// TIA Portal project "elektro_boiler" (V16)

(* hardware
DEVICE "S7-1200 station_1"  S7-1200 Station
   slot 0: "Rack_0"  S7-1200 Rack  Rack  V1.0
   slot 1: "PLC_1"  CPU 1215C DC/DC/Rly  6ES7 215-1HG40-0XB0  V4.4
   slot 2: "AI 8x13BIT_1"  6ES7 231-4HF32-0XB0  V2.1
*)

// ===== PLC "PLC_1"  CPU 1215C DC/DC/Rly =====

VAR_GLOBAL   // PLC tag table "Default tag table"
   "Clock_Byte" AT %MB0 : Byte;
   "Clock_10Hz" AT %M0.0 : Bool;
   "Clock_5Hz" AT %M0.1 : Bool;
   "Clock_2.5Hz" AT %M0.2 : Bool;
   "Clock_2Hz" AT %M0.3 : Bool;
   "Clock_1.25Hz" AT %M0.4 : Bool;
   "Clock_1Hz" AT %M0.5 : Bool;
   "Clock_0.625Hz" AT %M0.6 : Bool;
   "Clock_0.5Hz" AT %M0.7 : Bool;
   "TRUE" AT %M5.1 : Bool;
   "FALSE" AT %M5.0 : Bool;
   "puls_1_sec_t" AT %M4.0 : Bool;
   "puls_1_sec" AT %M4.1 : Bool;
   "EVEN" AT %M4.2 : Bool;
   "ODD" AT %M4.3 : Bool;
   "System_Byte" AT %MB1 : Byte;
   "FirstScan" AT %M1.0 : Bool;
   "DiagStatusUpdate" AT %M1.1 : Bool;
   "AlwaysTRUE" AT %M1.2 : Bool;
   "AlwaysFALSE" AT %M1.3 : Bool;
   "System_Byte(1)" AT %MB1 : Byte;
   "PUMP" AT %I0.0 : Bool;
   "AUTO_MAN" AT %I0.1 : Bool;
   "ELECTODE_DI1" AT %I0.2 : Bool;
   "ELECTODE_DI2" AT %I0.3 : Bool;
   "ELECTODE_DI3" AT %I0.4 : Bool;
   "ELECTODE_DI4" AT %I0.5 : Bool;
   "ELECTODE_DI5" AT %I0.6 : Bool;
   "ELECTODE_DI6" AT %I0.7 : Bool;
   "ELECTODE_DI7" AT %I1.0 : Bool;
   "ELECTODE_DI8" AT %I1.1 : Bool;
   "Tag_1" AT %Q1.1 : Bool;
   "Tag_2" AT %M6.0 : Bool;
END_VAR

VAR_GLOBAL   // PLC tag table "DO"
   "ELECTR_DO_1" AT %Q0.0 : Bool;
   "ELECTR_DO_2" AT %Q0.1 : Bool;
   "ELECTR_DO_3" AT %Q0.2 : Bool;
   "ELECTR_DO_4" AT %Q0.3 : Bool;
   "ELECTR_DO_5" AT %Q0.4 : Bool;
   "ELECTR_DO_6" AT %Q0.5 : Bool;
   "ELECTR_DO_7" AT %Q0.6 : Bool;
   "ELECTR_DO_8" AT %Q0.7 : Bool;
   "ZUMMER" AT %Q1.0 : Bool;
END_VAR

VAR_GLOBAL   // PLC tag table "AI"
   "PRESSURE" AT %IW112 : Int;
   "TEMP_IN" AT %IW114 : Int;
   "res1" AT %IW116 : Int;
   "CURRENT_A" AT %IW118 : Int;
   "CURRENT_B" AT %IW120 : Int;
   "CURRENT_C" AT %IW122 : Int;
END_VAR

TYPE "AIN"
   STRUCT
      data_raw : Int;   // Сырое значение
      signal : Real;   // Значение сигнала в электрических единицах (мА, В и т.д.)
      eng : Real;   // Масштабированное значение аналогового сигнала
      status_0 : Bool;   // Неисправность канала
      status_1 : Bool;   // Ошибка калибровки (CalFault)
      status_2 : Bool;   // Выше HH
      status_3 : Bool;   // Выше H
      status_4 : Bool;   // Ниже L
      status_5 : Bool;   // Ниже LL
      status_6 : Bool;   // Резерв.
      status_7 : Bool;   // Выше диапазона (OverRange)
      status_8 : Bool;   // Ниже диапазона (UnderRange
      status_9 : Bool;   // Выше шкалы (OverScale)
      status_10 : Bool;   // Ниже шкалы (UnderScale)
      status_11 : Bool;   // Резерв.
      status_12 : Bool;   // Резерв.
      status_13 : Bool;   // Резерв.
      status_14 : Bool;   // Маскирование сигнала включено
      status_15 : Bool;   // Имитация сигнала включена
      SclMax : Real;   // Максимальное значение шкалы сигнала (в инженерных
      SclMin : Real;   // Минимальное значение шкалы сигнала (в инженерных
      DeadBand : Real;   // Значение уставки зоны нечувствительности (в инженерных
      LL : Real;   // Значение уставки LL (в инженерных единицах)
      L : Real;   // Значение уставки L (в инженерных единицах)
      H : Real := 90.0;   // Значение уставки H (в инженерных единицах)
      HH : Real := 100.0;   // Значение уставки HH (в инженерных единицах)
      config_0 : Bool;   // Команда: включить имитацию аналогового сигнала
      config_1 : Bool;   // Зарезервировано
      config_2 : Bool;   // Команда: включить в обработку уставку LL
      config_3 : Bool;   // Команда: включить в обработку уставку L
      config_4 : Bool;   // Команда: включить в обработку уставку H
      config_5 : Bool;   // Команда: включить в обработку уставку HH
      config_6 : Bool;   // Зарезервировано
      config_7 : Bool;   // Не используется
      config_8 : Bool;   // Команда: включить маскирование сигнала
      descID : Int;   // ID описания
   END_STRUCT;
END_TYPE

DATA_BLOCK "HMI"   // DB1
{ S7_Optimized_Access := 'FALSE' }
VERSION : 0.1
   VAR
      PUMP_STOP : Bool;
      HI_PRESSURE : Bool;
      FAIL_EL1 : Bool;
      FAIL_EL2 : Bool;
      FAIL_EL3 : Bool;
      FAIL_EL4 : Bool;
      FAIL_EL5 : Bool;
      FAIL_EL6 : Bool;
      FAIL_EL7 : Bool;
      FAIL_EL8 : Bool;
      ACKNOWLEDGE : Bool;
      ELEC_OFF1 : Bool;
      ELEC_OFF2 : Bool;
      ELEC_OFF3 : Bool;
      ELEC_OFF4 : Bool;
      ELEC_OFF5 : Bool;
      ELEC_OFF6 : Bool;
      ELEC_OFF7 : Bool;
      ELEC_OFF8 : Bool;
      DO_TEST : Bool;
      T_SIMUL : Bool;
      P_SIMUL : Bool;
      T_NO_SIG : Bool;
      P_NO_SIG : Bool;
      T_OVERSCALE : Bool;
      P_OVERSCALE : Bool;
      reserv7 : Bool;
      reserv8 : Bool;
      reserv9 : Bool;
      reserv10 : Bool;
      reserv11 : Bool;
      reserv12 : Bool;
      T_MAX : Int := 1500;
      T_MIIN : Int := -500;
      T_DREYF : Int;
      T_SP : Int := 600;
      T_PV : Int;
      T_DELTA : Int := 10;
      P_MAX : Int := 60;
      P_MIIN : Int;
      P_DREYF : Int;
      P_PV : Int := 40;
      P_ALARM : Int;
      P_DELTA : Int := 10;
      CHANGE_TIME : Int := 3600;
      T_SIM_VAL : Int;
      P_SIM_VAL : Int;
   END_VAR
BEGIN
END_DATA_BLOCK

DATA_BLOCK "TEMP_DB"   // DB2
{ S7_Optimized_Access := 'TRUE' }
VERSION : 0.1
   VAR
      RESET_DO_TEST : TON_TIME;
      GEN_ALAR : Bool;
      T_CHANGE : Time := T#2s;
      ET3 : DWord;
      ET4 : DWord;
      ET5 : DWord;
      ET6 : DWord;
      ET7 : DWord;
      ET8 : DWord;
      WARNING : Bool;
   END_VAR
BEGIN
END_DATA_BLOCK

DATA_BLOCK "MB_Config"   // DB3
{ S7_Optimized_Access := 'TRUE' }
VERSION : 0.1
   VAR
      HOLD_REG : Array[0..49] of Int;
      CONNECT : TCON_IP_v4;
      ERROR : Bool;
      STATUS : Word;
      DISCONNECT : Bool;
      MODE : USInt := 1;
      DATA_ADDR : UDInt := 40001;
      DATA_LEN : UDInt := 10;
      DONE : Bool;
      BUSY : Bool;
   END_VAR
BEGIN
   CONNECT.RemotePort := 102;
   CONNECT.RemoteAddress.ADDR[4] := 2;
   CONNECT.RemoteAddress.ADDR[3] := 1;
   CONNECT.RemoteAddress.ADDR[2] := 168;
   CONNECT.RemoteAddress.ADDR[1] := 192;
   CONNECT.ActiveEstablished := true;
   CONNECT.ConnectionType := 11;
   CONNECT.ID := 1;
   CONNECT.InterfaceId := 64;
END_DATA_BLOCK

DATA_BLOCK "BUFFER"   // DB5
{ S7_Optimized_Access := 'FALSE' }
VERSION : 0.1
   VAR
      DATA : Array[0..20] of Word;
   END_VAR
BEGIN
   DATA[4] := -500;   // T_MIN
   DATA[5] := 0;   // T_DREYF
   DATA[6] := 600;   // T_SP
   DATA[8] := 10;   // T_DELTA
   DATA[9] := 60;   // P_MAX
   DATA[10] := 0;   // P_MIIN
   DATA[11] := 0;   // P_DREYF
   DATA[3] := 1500;   // T_MAX
   DATA[12] := 0;   // P_PV
   DATA[13] := 40;   // P_ALARM
   DATA[14] := 0;   // P_DELTA
   DATA[15] := 3600;   // CHANGE_TIME
   DATA[16] := 200;   // T_SIM_VAL
   DATA[17] := 300;   // P_SIM_VAL
   // DATA[7] : T_PV
END_DATA_BLOCK

FUNCTION "AINS_general" : Void   // FC1, SCL
{ S7_Optimized_Access := 'TRUE' }
VERSION : 0.1
   VAR_INPUT
      MAX : Int;
      MIN : Int;
      DREYF : Int;
      ANALOG_IN_PUT : Int;
      SIMUL_VAL : Int;
      SIMUL_ENAB : Bool;
   END_VAR
   VAR_OUTPUT
      ANALOG_OUT_PUT : Int;
      NO_SIGNAL : Bool;
      OVER_SCLAE : Bool;
   END_VAR
   VAR_TEMP
      TMP1 : Real;
      TMP2 : Real;
      TMP3 : Int;
   END_VAR
BEGIN
   IF (#SIMUL_ENAB = FALSE) THEN
       #TMP1 := INT_TO_REAL(#MAX - #MIN) / 10.0;
       #TMP1 := #TMP1 * INT_TO_REAL(#ANALOG_IN_PUT);
       #TMP2 := #TMP1 / 27648.0;
       #TMP3 := REAL_TO_INT(#TMP2 * 10) + #MIN;

       #NO_SIGNAL := (#ANALOG_IN_PUT = 32767);
       #OVER_SCLAE := (#ANALOG_IN_PUT > 27648) AND NOT #NO_SIGNAL;
       IF (NOT #NO_SIGNAL) THEN
           #ANALOG_OUT_PUT := #TMP3 + #DREYF;
       ELSE
           #ANALOG_OUT_PUT := 0;
       END_IF;
   ELSE
       #ANALOG_OUT_PUT := #SIMUL_VAL;
   END_IF;
END_FUNCTION

FUNCTION "AINS_main" : Void   // FC2, LAD
{ S7_Optimized_Access := 'TRUE' }
VERSION : 0.1
BEGIN

REGION Network 1
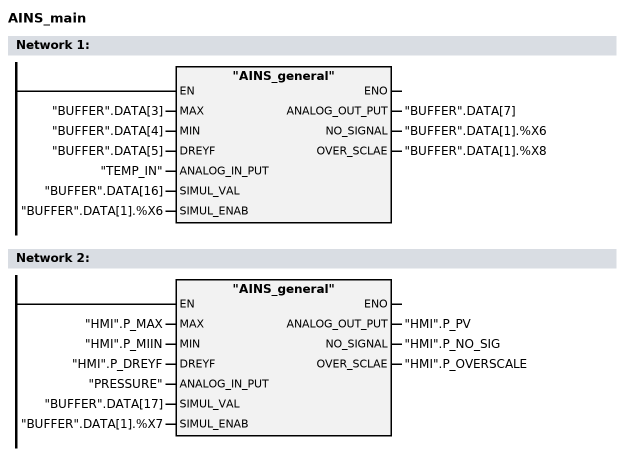
   RUNG wire#powerrail
      "AINS_general"(MAX := "BUFFER".DATA[3], MIN := "BUFFER".DATA[4], DREYF := "BUFFER".DATA[5], ANALOG_IN_PUT := "TEMP_IN", SIMUL_VAL := "BUFFER".DATA[16], SIMUL_ENAB := "BUFFER".DATA[1].%X6, ANALOG_OUT_PUT => "BUFFER".DATA[7], NO_SIGNAL => "BUFFER".DATA[1].%X6, OVER_SCLAE => "BUFFER".DATA[1].%X8)
   END_RUNG
   // the same network as SCL:
   "AINS_general"(MAX := "BUFFER".DATA[3],
                  MIN := "BUFFER".DATA[4],
                  DREYF := "BUFFER".DATA[5],
                  ANALOG_IN_PUT := "TEMP_IN",
                  SIMUL_VAL := "BUFFER".DATA[16],
                  SIMUL_ENAB := "BUFFER".DATA[1].%X6,
                  ANALOG_OUT_PUT => "BUFFER".DATA[7],
                  NO_SIGNAL => "BUFFER".DATA[1].%X6,
                  OVER_SCLAE => "BUFFER".DATA[1].%X8);
END_REGION

REGION Network 2
   RUNG wire#powerrail
      "AINS_general"(MAX := "HMI".P_MAX, MIN := "HMI".P_MIIN, DREYF := "HMI".P_DREYF, ANALOG_IN_PUT := "PRESSURE", SIMUL_VAL := "BUFFER".DATA[17], SIMUL_ENAB := "BUFFER".DATA[1].%X7, ANALOG_OUT_PUT => "HMI".P_PV, NO_SIGNAL => "HMI".P_NO_SIG, OVER_SCLAE => "HMI".P_OVERSCALE)
   END_RUNG
   // the same network as SCL:
   "AINS_general"(MAX := "HMI".P_MAX,
                  MIN := "HMI".P_MIIN,
                  DREYF := "HMI".P_DREYF,
                  ANALOG_IN_PUT := "PRESSURE",
                  SIMUL_VAL := "BUFFER".DATA[17],
                  SIMUL_ENAB := "BUFFER".DATA[1].%X7,
                  ANALOG_OUT_PUT => "HMI".P_PV,
                  NO_SIGNAL => "HMI".P_NO_SIG,
                  OVER_SCLAE => "HMI".P_OVERSCALE);
END_REGION
END_FUNCTION

FUNCTION "Chang_general" : Void   // FC3, LAD
{ S7_Optimized_Access := 'TRUE' }
VERSION : 0.1
   VAR_INPUT
      SEKUNDS : DWord;
   END_VAR
   VAR_OUTPUT
      FIRST : Bool;
      SECOND : Bool;
   END_VAR
   VAR_TEMP
      SECOND_time : DWord;
      TMP : DWord;
   END_VAR
BEGIN

REGION Network 1
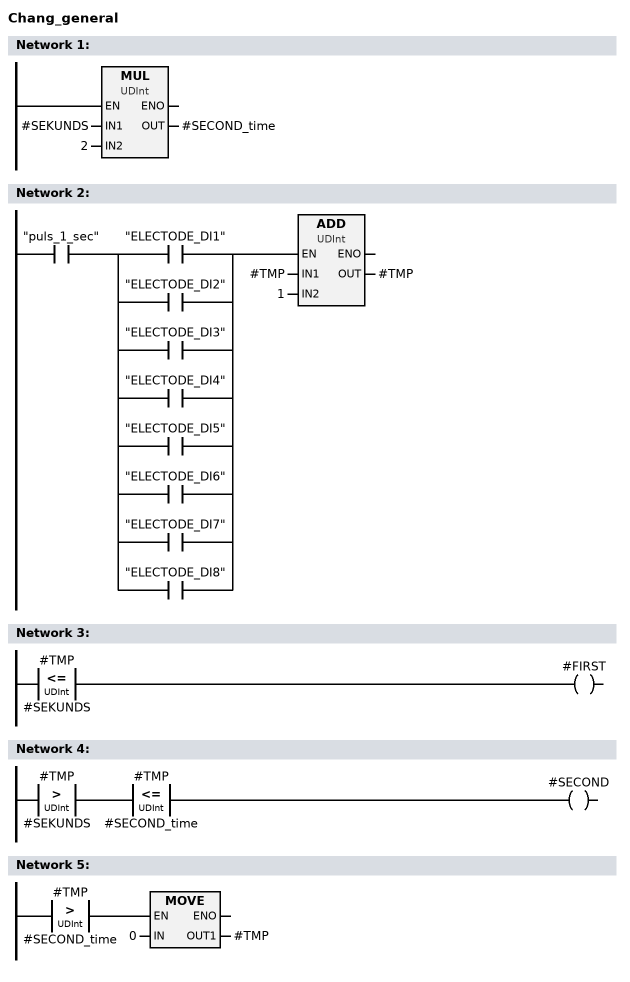
   RUNG wire#powerrail
      { S7_Templates := "SrcType := UDInt" } Mul(in1 := #SEKUNDS, in2 := 2, out => #SECOND_time)
   END_RUNG
   // the same network as SCL:
   #SECOND_time := #SEKUNDS * 2;
END_REGION

REGION Network 2
   RUNG wire#powerrail
      Contact( "puls_1_sec" )
      wire#w1
      Contact( "ELECTODE_DI1" )
      wire#w2
      { S7_Templates := "SrcType := UDInt" } Add(in1 := #TMP, in2 := 1, out => #TMP)
   END_RUNG
   RUNG wire#w1
      Contact( "ELECTODE_DI2" )
   END_RUNG wire#w2
   RUNG wire#w1
      Contact( "ELECTODE_DI3" )
   END_RUNG wire#w2
   RUNG wire#w1
      Contact( "ELECTODE_DI4" )
   END_RUNG wire#w2
   RUNG wire#w1
      Contact( "ELECTODE_DI5" )
   END_RUNG wire#w2
   RUNG wire#w1
      Contact( "ELECTODE_DI6" )
   END_RUNG wire#w2
   RUNG wire#w1
      Contact( "ELECTODE_DI7" )
   END_RUNG wire#w2
   RUNG wire#w1
      Contact( "ELECTODE_DI8" )
   END_RUNG wire#w2
   // the same network as SCL:
   IF "puls_1_sec" AND ("ELECTODE_DI1" OR "ELECTODE_DI2" OR "ELECTODE_DI3" OR "ELECTODE_DI4" OR "ELECTODE_DI5" OR "ELECTODE_DI6" OR "ELECTODE_DI7" OR "ELECTODE_DI8") THEN
       #TMP := #TMP + 1;
   END_IF;
END_REGION

REGION Network 3
   RUNG wire#powerrail
      { S7_Templates := "SrcType := UDInt" } LE_Contact(in1 := #TMP, in2 := #SEKUNDS)
      Coil( #FIRST )
   END_RUNG
   // the same network as SCL:
   #FIRST := #TMP <= #SEKUNDS;
END_REGION

REGION Network 4
   RUNG wire#powerrail
      { S7_Templates := "SrcType := UDInt" } GT_Contact(in1 := #TMP, in2 := #SEKUNDS)
      { S7_Templates := "SrcType := UDInt" } LE_Contact(in1 := #TMP, in2 := #SECOND_time)
      Coil( #SECOND )
   END_RUNG
   // the same network as SCL:
   #SECOND := (#TMP > #SEKUNDS) AND (#TMP <= #SECOND_time);
END_REGION

REGION Network 5
   RUNG wire#powerrail
      { S7_Templates := "SrcType := UDInt" } GT_Contact(in1 := #TMP, in2 := #SECOND_time)
      Move(in := 0, out1 => #TMP)
   END_RUNG
   // the same network as SCL:
   IF #TMP > #SECOND_time THEN #TMP := 0; END_IF;
END_REGION
END_FUNCTION

FUNCTION "Cange_main" : Void   // FC4, LAD
{ S7_Optimized_Access := 'TRUE' }
VERSION : 0.1
   VAR_TEMP
      TTT : Time;
   END_VAR
BEGIN

REGION Network 1
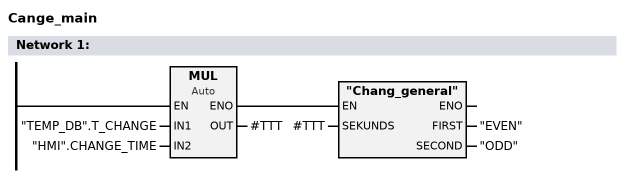
   RUNG wire#powerrail
      Mul(in1 := "TEMP_DB".T_CHANGE, in2 := "HMI".CHANGE_TIME, out => #TTT)
      "Chang_general"(SEKUNDS := #TTT, FIRST => "EVEN", SECOND => "ODD")
   END_RUNG
   // the same network as SCL:
   #TTT := "TEMP_DB".T_CHANGE * "HMI".CHANGE_TIME;
   "Chang_general"(SEKUNDS := #TTT, FIRST => "EVEN", SECOND => "ODD");
END_REGION
END_FUNCTION

FUNCTION "DOUT_general" : Void   // FC5, LAD
{ S7_Optimized_Access := 'TRUE' }
VERSION : 0.1
   VAR_INPUT
      AIN : Real;
      SET_POINT : Real;
      DEADBAND : Real;
   END_VAR
   VAR_OUTPUT
      OUT : Bool;
   END_VAR
   VAR_TEMP
      TEMPR_MIN : Real;
      TEMPR_MAX : Real;
   END_VAR
BEGIN

REGION Network 1
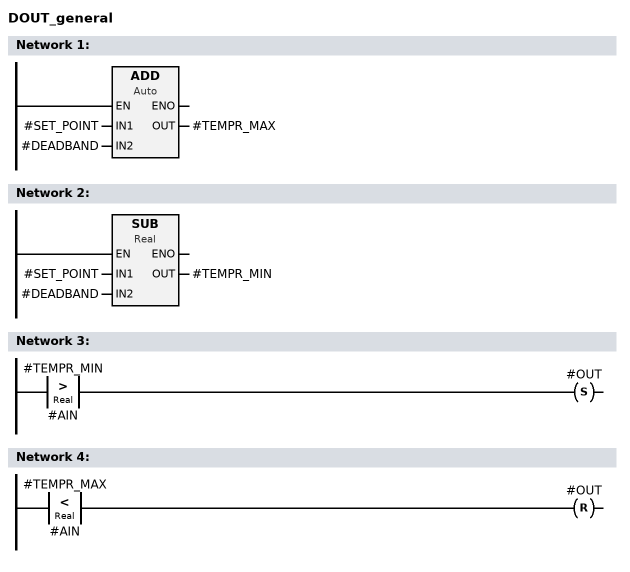
   RUNG wire#powerrail
      Add(in1 := #SET_POINT, in2 := #DEADBAND, out => #TEMPR_MAX)
   END_RUNG
   // the same network as SCL:
   #TEMPR_MAX := #SET_POINT + #DEADBAND;
END_REGION

REGION Network 2
   RUNG wire#powerrail
      { S7_Templates := "SrcType := Real" } Sub(in1 := #SET_POINT, in2 := #DEADBAND, out => #TEMPR_MIN)
   END_RUNG
   // the same network as SCL:
   #TEMPR_MIN := #SET_POINT - #DEADBAND;
END_REGION

REGION Network 3
   RUNG wire#powerrail
      { S7_Templates := "SrcType := Real" } GT_Contact(in1 := #TEMPR_MIN, in2 := #AIN)
      S_Coil( #OUT )
   END_RUNG
   // the same network as SCL:
   IF #TEMPR_MIN > #AIN THEN #OUT := TRUE; END_IF;
END_REGION

REGION Network 4
   RUNG wire#powerrail
      { S7_Templates := "SrcType := Real" } LT_Contact(in1 := #TEMPR_MAX, in2 := #AIN)
      R_Coil( #OUT )
   END_RUNG
   // the same network as SCL:
   IF #TEMPR_MAX < #AIN THEN #OUT := FALSE; END_IF;
END_REGION
END_FUNCTION

FUNCTION "DOUT_main" : Void   // FC6, LAD
{ S7_Optimized_Access := 'TRUE' }
VERSION : 0.1
   VAR_TEMP
      OUT : Bool;
   END_VAR
   VAR_TEMP   // added for the SCL form of the ladder/FBD networks
      _w1 : Bool;
   END_VAR
BEGIN

REGION Network 1
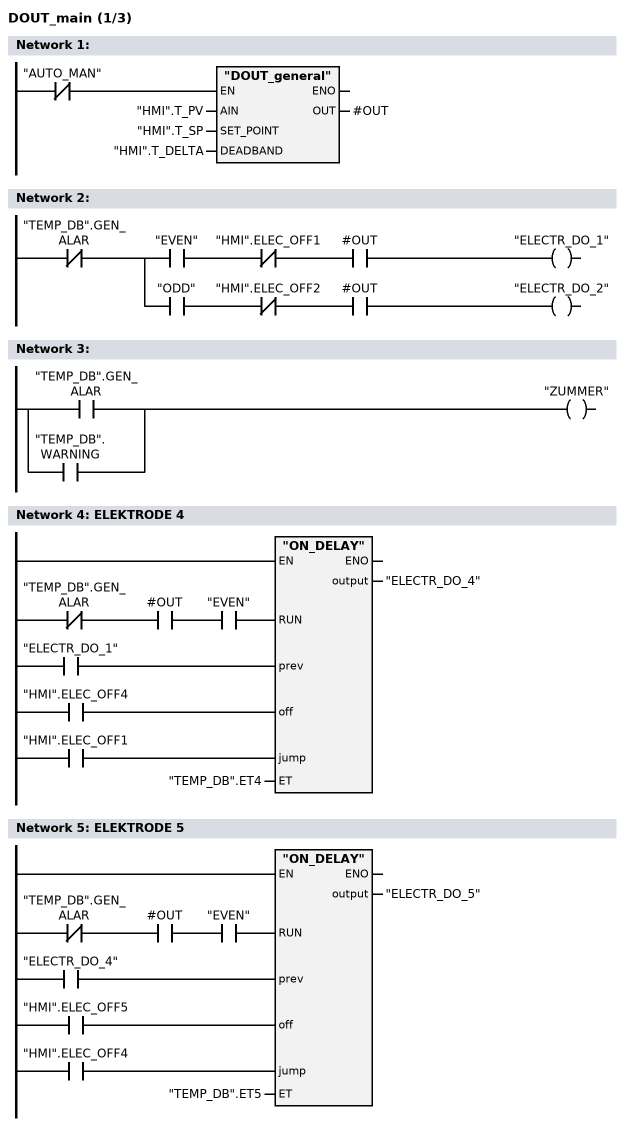
   RUNG wire#powerrail
      I_Contact( "AUTO_MAN" )
      "DOUT_general"(AIN := "HMI".T_PV, SET_POINT := "HMI".T_SP, DEADBAND := "HMI".T_DELTA, OUT => #OUT)
   END_RUNG
   // the same network as SCL:
   IF NOT "AUTO_MAN" THEN
       "DOUT_general"(AIN := "HMI".T_PV, SET_POINT := "HMI".T_SP, DEADBAND := "HMI".T_DELTA, OUT => #OUT);
   END_IF;
END_REGION

REGION Network 2
   RUNG wire#powerrail
      I_Contact( "TEMP_DB".GEN_ALAR )
      wire#w1
      Contact( "EVEN" )
      I_Contact( "HMI".ELEC_OFF1 )
      Contact( #OUT )
      Coil( "ELECTR_DO_1" )
   END_RUNG
   RUNG wire#w1
      Contact( "ODD" )
      I_Contact( "HMI".ELEC_OFF2 )
      Contact( #OUT )
      Coil( "ELECTR_DO_2" )
   END_RUNG
   // the same network as SCL:
   "ELECTR_DO_1" := NOT "TEMP_DB".GEN_ALAR AND "EVEN" AND NOT "HMI".ELEC_OFF1 AND #OUT;
   "ELECTR_DO_2" := NOT "TEMP_DB".GEN_ALAR AND "ODD" AND NOT "HMI".ELEC_OFF2 AND #OUT;
END_REGION

REGION Network 3
   RUNG wire#powerrail
      Contact( "TEMP_DB".GEN_ALAR )
      wire#w1
      Coil( "ZUMMER" )
   END_RUNG
   RUNG wire#powerrail
      Contact( "TEMP_DB".WARNING )
   END_RUNG wire#w1
   // the same network as SCL:
   "ZUMMER" := "TEMP_DB".GEN_ALAR OR "TEMP_DB".WARNING;
END_REGION

REGION Network 4: ELEKTRODE 4
   RUNG wire#powerrail
      "ON_DELAY"(RUN := wire#w1, prev := wire#w2, off := wire#w3, jump := wire#w4, ET := "TEMP_DB".ET4, output => "ELECTR_DO_4")
   END_RUNG
   RUNG wire#powerrail
      I_Contact( "TEMP_DB".GEN_ALAR )
      Contact( #OUT )
      Contact( "EVEN" )
   END_RUNG wire#w1
   RUNG wire#powerrail
      Contact( "ELECTR_DO_1" )
   END_RUNG wire#w2
   RUNG wire#powerrail
      Contact( "HMI".ELEC_OFF4 )
   END_RUNG wire#w3
   RUNG wire#powerrail
      Contact( "HMI".ELEC_OFF1 )
   END_RUNG wire#w4
   // the same network as SCL:
   "ON_DELAY"(RUN := NOT "TEMP_DB".GEN_ALAR AND #OUT AND "EVEN",
              prev := "ELECTR_DO_1",
              off := "HMI".ELEC_OFF4,
              jump := "HMI".ELEC_OFF1,
              ET := "TEMP_DB".ET4,
              output => "ELECTR_DO_4");
END_REGION

REGION Network 5: ELEKTRODE 5
   RUNG wire#powerrail
      "ON_DELAY"(RUN := wire#w1, prev := wire#w2, off := wire#w3, jump := wire#w4, ET := "TEMP_DB".ET5, output => "ELECTR_DO_5")
   END_RUNG
   RUNG wire#powerrail
      I_Contact( "TEMP_DB".GEN_ALAR )
      Contact( #OUT )
      Contact( "EVEN" )
   END_RUNG wire#w1
   RUNG wire#powerrail
      Contact( "ELECTR_DO_4" )
   END_RUNG wire#w2
   RUNG wire#powerrail
      Contact( "HMI".ELEC_OFF5 )
   END_RUNG wire#w3
   RUNG wire#powerrail
      Contact( "HMI".ELEC_OFF4 )
   END_RUNG wire#w4
   // the same network as SCL:
   "ON_DELAY"(RUN := NOT "TEMP_DB".GEN_ALAR AND #OUT AND "EVEN",
              prev := "ELECTR_DO_4",
              off := "HMI".ELEC_OFF5,
              jump := "HMI".ELEC_OFF4,
              ET := "TEMP_DB".ET5,
              output => "ELECTR_DO_5");
END_REGION

REGION Network 6: ELEKTRODE 8
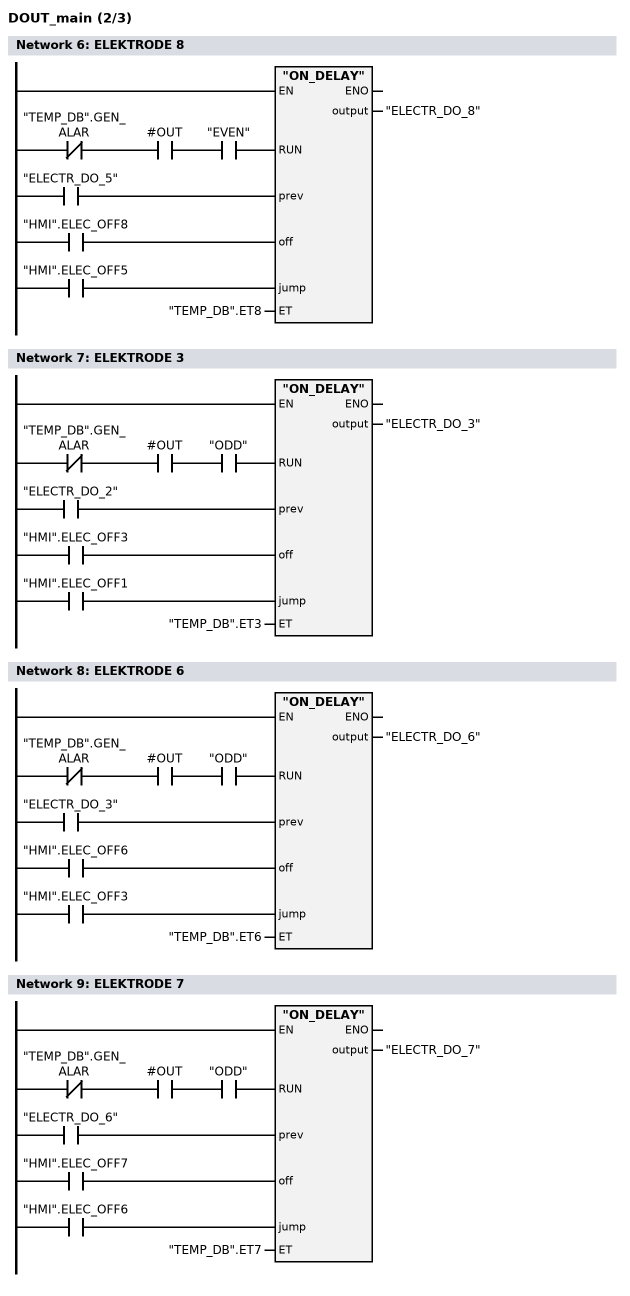
   RUNG wire#powerrail
      "ON_DELAY"(RUN := wire#w1, prev := wire#w2, off := wire#w3, jump := wire#w4, ET := "TEMP_DB".ET8, output => "ELECTR_DO_8")
   END_RUNG
   RUNG wire#powerrail
      I_Contact( "TEMP_DB".GEN_ALAR )
      Contact( #OUT )
      Contact( "EVEN" )
   END_RUNG wire#w1
   RUNG wire#powerrail
      Contact( "ELECTR_DO_5" )
   END_RUNG wire#w2
   RUNG wire#powerrail
      Contact( "HMI".ELEC_OFF8 )
   END_RUNG wire#w3
   RUNG wire#powerrail
      Contact( "HMI".ELEC_OFF5 )
   END_RUNG wire#w4
   // the same network as SCL:
   "ON_DELAY"(RUN := NOT "TEMP_DB".GEN_ALAR AND #OUT AND "EVEN",
              prev := "ELECTR_DO_5",
              off := "HMI".ELEC_OFF8,
              jump := "HMI".ELEC_OFF5,
              ET := "TEMP_DB".ET8,
              output => "ELECTR_DO_8");
END_REGION

REGION Network 7: ELEKTRODE 3
   RUNG wire#powerrail
      "ON_DELAY"(RUN := wire#w1, prev := wire#w2, off := wire#w3, jump := wire#w4, ET := "TEMP_DB".ET3, output => "ELECTR_DO_3")
   END_RUNG
   RUNG wire#powerrail
      I_Contact( "TEMP_DB".GEN_ALAR )
      Contact( #OUT )
      Contact( "ODD" )
   END_RUNG wire#w1
   RUNG wire#powerrail
      Contact( "ELECTR_DO_2" )
   END_RUNG wire#w2
   RUNG wire#powerrail
      Contact( "HMI".ELEC_OFF3 )
   END_RUNG wire#w3
   RUNG wire#powerrail
      Contact( "HMI".ELEC_OFF1 )
   END_RUNG wire#w4
   // the same network as SCL:
   "ON_DELAY"(RUN := NOT "TEMP_DB".GEN_ALAR AND #OUT AND "ODD",
              prev := "ELECTR_DO_2",
              off := "HMI".ELEC_OFF3,
              jump := "HMI".ELEC_OFF1,
              ET := "TEMP_DB".ET3,
              output => "ELECTR_DO_3");
END_REGION

REGION Network 8: ELEKTRODE 6
   RUNG wire#powerrail
      "ON_DELAY"(RUN := wire#w1, prev := wire#w2, off := wire#w3, jump := wire#w4, ET := "TEMP_DB".ET6, output => "ELECTR_DO_6")
   END_RUNG
   RUNG wire#powerrail
      I_Contact( "TEMP_DB".GEN_ALAR )
      Contact( #OUT )
      Contact( "ODD" )
   END_RUNG wire#w1
   RUNG wire#powerrail
      Contact( "ELECTR_DO_3" )
   END_RUNG wire#w2
   RUNG wire#powerrail
      Contact( "HMI".ELEC_OFF6 )
   END_RUNG wire#w3
   RUNG wire#powerrail
      Contact( "HMI".ELEC_OFF3 )
   END_RUNG wire#w4
   // the same network as SCL:
   "ON_DELAY"(RUN := NOT "TEMP_DB".GEN_ALAR AND #OUT AND "ODD",
              prev := "ELECTR_DO_3",
              off := "HMI".ELEC_OFF6,
              jump := "HMI".ELEC_OFF3,
              ET := "TEMP_DB".ET6,
              output => "ELECTR_DO_6");
END_REGION

REGION Network 9: ELEKTRODE 7
   RUNG wire#powerrail
      "ON_DELAY"(RUN := wire#w1, prev := wire#w2, off := wire#w3, jump := wire#w4, ET := "TEMP_DB".ET7, output => "ELECTR_DO_7")
   END_RUNG
   RUNG wire#powerrail
      I_Contact( "TEMP_DB".GEN_ALAR )
      Contact( #OUT )
      Contact( "ODD" )
   END_RUNG wire#w1
   RUNG wire#powerrail
      Contact( "ELECTR_DO_6" )
   END_RUNG wire#w2
   RUNG wire#powerrail
      Contact( "HMI".ELEC_OFF7 )
   END_RUNG wire#w3
   RUNG wire#powerrail
      Contact( "HMI".ELEC_OFF6 )
   END_RUNG wire#w4
   // the same network as SCL:
   "ON_DELAY"(RUN := NOT "TEMP_DB".GEN_ALAR AND #OUT AND "ODD",
              prev := "ELECTR_DO_6",
              off := "HMI".ELEC_OFF7,
              jump := "HMI".ELEC_OFF6,
              ET := "TEMP_DB".ET7,
              output => "ELECTR_DO_7");
END_REGION

REGION Network 10
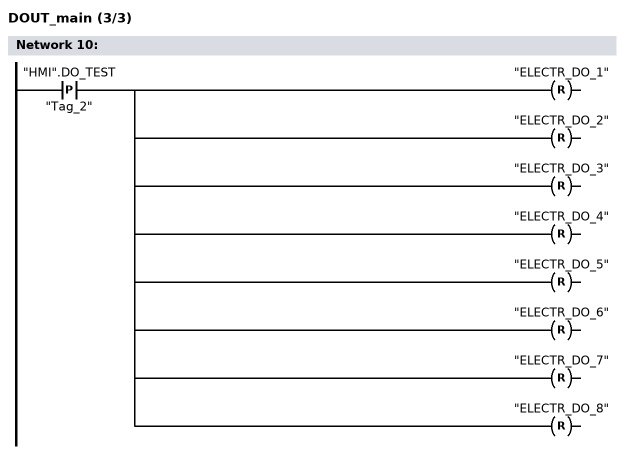
   RUNG wire#powerrail
      P_Contact(operand := "HMI".DO_TEST, bit := "Tag_2")
      wire#w1
      R_Coil( "ELECTR_DO_1" )
   END_RUNG
   RUNG wire#w1
      R_Coil( "ELECTR_DO_2" )
   END_RUNG
   RUNG wire#w1
      R_Coil( "ELECTR_DO_3" )
   END_RUNG
   RUNG wire#w1
      R_Coil( "ELECTR_DO_4" )
   END_RUNG
   RUNG wire#w1
      R_Coil( "ELECTR_DO_5" )
   END_RUNG
   RUNG wire#w1
      R_Coil( "ELECTR_DO_6" )
   END_RUNG
   RUNG wire#w1
      R_Coil( "ELECTR_DO_7" )
   END_RUNG
   RUNG wire#w1
      R_Coil( "ELECTR_DO_8" )
   END_RUNG
   // the same network as SCL:
   #_w1 := "HMI".DO_TEST AND NOT "Tag_2";   // rising edge of "HMI".DO_TEST
   "Tag_2" := "HMI".DO_TEST;
   IF #_w1 THEN
       "ELECTR_DO_1" := FALSE;
       "ELECTR_DO_2" := FALSE;
       "ELECTR_DO_3" := FALSE;
       "ELECTR_DO_4" := FALSE;
       "ELECTR_DO_5" := FALSE;
       "ELECTR_DO_6" := FALSE;
       "ELECTR_DO_7" := FALSE;
       "ELECTR_DO_8" := FALSE;
   END_IF;
END_REGION
END_FUNCTION

FUNCTION "AINS_general_1" : Void   // FC7, SCL
{ S7_Optimized_Access := 'TRUE' }
VERSION : 0.1
   VAR_INPUT
      MAX : Real;
      MIN : Real;
      DREYF : Real;
      ANALOG_IN_PUT : Int;
   END_VAR
   VAR_OUTPUT
      ANALOG_OUT_PUT : Real;
   END_VAR
   VAR_TEMP
      TMP1 : DInt;
      TMP2 : Real;
   END_VAR
BEGIN
   #TMP1 := REAL_TO_DINT(#MAX - #MIN);
   #TMP1 := #TMP1 * #ANALOG_IN_PUT;
   #TMP2 := DINT_TO_REAL(#TMP1) / 27648.0;
   #TMP2 := #TMP2 + #MIN;
   #ANALOG_OUT_PUT := #TMP2 + #DREYF;
END_FUNCTION

FUNCTION "ON_DELAY" : Void   // FC8, LAD
{ S7_Optimized_Access := 'TRUE' }
VERSION : 0.1
   VAR_INPUT
      RUN : Bool;
      prev : Bool;
      off : Bool;
      jump : Bool;
   END_VAR
   VAR_OUTPUT
      output : Bool;
   END_VAR
   VAR_IN_OUT
      ET : DWord;
   END_VAR
   VAR_TEMP
      RRRR : Bool;
   END_VAR
BEGIN

REGION Network 1
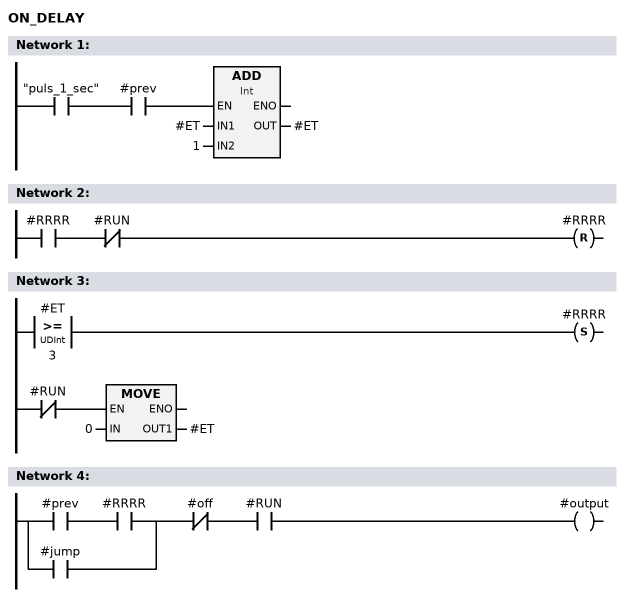
   RUNG wire#powerrail
      Contact( "puls_1_sec" )
      Contact( #prev )
      { S7_Templates := "SrcType := Int" } Add(in1 := #ET, in2 := 1, out => #ET)
   END_RUNG
   // the same network as SCL:
   IF "puls_1_sec" AND #prev THEN #ET := #ET + 1; END_IF;
END_REGION

REGION Network 2
   RUNG wire#powerrail
      Contact( #RRRR )
      I_Contact( #RUN )
      R_Coil( #RRRR )
   END_RUNG
   // the same network as SCL:
   IF #RRRR AND NOT #RUN THEN #RRRR := FALSE; END_IF;
END_REGION

REGION Network 3
   RUNG wire#powerrail
      { S7_Templates := "SrcType := UDInt" } GE_Contact(in1 := #ET, in2 := 3)
      S_Coil( #RRRR )
   END_RUNG
   RUNG wire#powerrail
      I_Contact( #RUN )
      Move(in := 0, out1 => #ET)
   END_RUNG
   // the same network as SCL:
   IF #ET >= 3 THEN #RRRR := TRUE; END_IF;
   IF NOT #RUN THEN #ET := 0; END_IF;
END_REGION

REGION Network 4
   RUNG wire#powerrail
      Contact( #prev )
      Contact( #RRRR )
      wire#w1
      I_Contact( #off )
      Contact( #RUN )
      Coil( #output )
   END_RUNG
   RUNG wire#powerrail
      Contact( #jump )
   END_RUNG wire#w1
   // the same network as SCL:
   #output := ((#prev AND #RRRR) OR #jump) AND NOT #off AND #RUN;
END_REGION
END_FUNCTION

FUNCTION "ALARMS_general" : Void   // FC9, LAD
{ S7_Optimized_Access := 'TRUE' }
VERSION : 0.1
BEGIN

REGION Network 1: HIGH PRESSURE ALARM
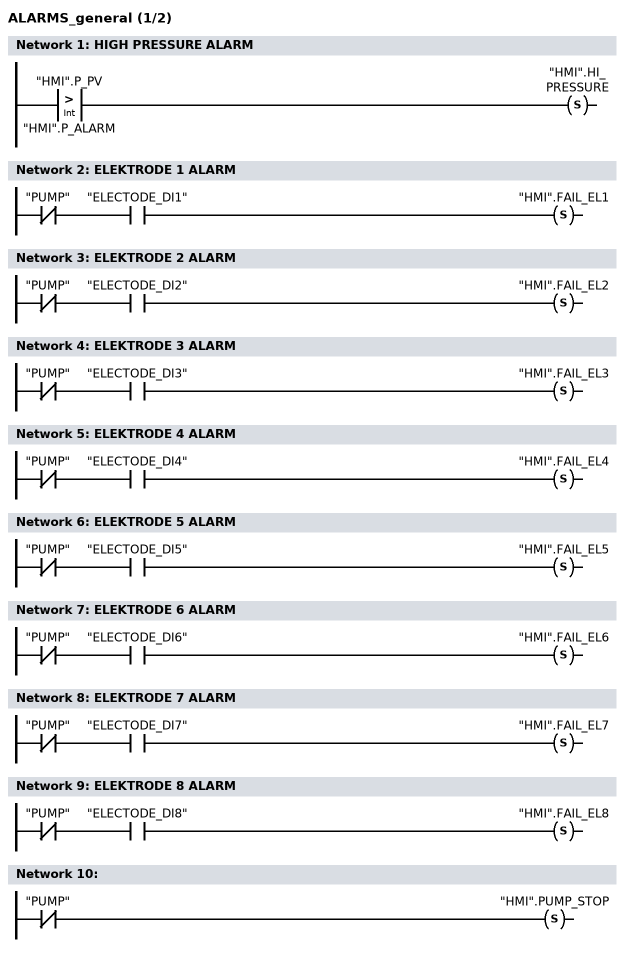
   RUNG wire#powerrail
      { S7_Templates := "SrcType := Int" } GT_Contact(in1 := "HMI".P_PV, in2 := "HMI".P_ALARM)
      S_Coil( "HMI".HI_PRESSURE )
   END_RUNG
   // the same network as SCL:
   IF "HMI".P_PV > "HMI".P_ALARM THEN "HMI".HI_PRESSURE := TRUE; END_IF;
END_REGION

REGION Network 2: ELEKTRODE 1 ALARM
   RUNG wire#powerrail
      I_Contact( "PUMP" )
      Contact( "ELECTODE_DI1" )
      S_Coil( "HMI".FAIL_EL1 )
   END_RUNG
   // the same network as SCL:
   IF NOT "PUMP" AND "ELECTODE_DI1" THEN "HMI".FAIL_EL1 := TRUE; END_IF;
END_REGION

REGION Network 3: ELEKTRODE 2 ALARM
   RUNG wire#powerrail
      I_Contact( "PUMP" )
      Contact( "ELECTODE_DI2" )
      S_Coil( "HMI".FAIL_EL2 )
   END_RUNG
   // the same network as SCL:
   IF NOT "PUMP" AND "ELECTODE_DI2" THEN "HMI".FAIL_EL2 := TRUE; END_IF;
END_REGION

REGION Network 4: ELEKTRODE 3 ALARM
   RUNG wire#powerrail
      I_Contact( "PUMP" )
      Contact( "ELECTODE_DI3" )
      S_Coil( "HMI".FAIL_EL3 )
   END_RUNG
   // the same network as SCL:
   IF NOT "PUMP" AND "ELECTODE_DI3" THEN "HMI".FAIL_EL3 := TRUE; END_IF;
END_REGION

REGION Network 5: ELEKTRODE 4 ALARM
   RUNG wire#powerrail
      I_Contact( "PUMP" )
      Contact( "ELECTODE_DI4" )
      S_Coil( "HMI".FAIL_EL4 )
   END_RUNG
   // the same network as SCL:
   IF NOT "PUMP" AND "ELECTODE_DI4" THEN "HMI".FAIL_EL4 := TRUE; END_IF;
END_REGION

REGION Network 6: ELEKTRODE 5 ALARM
   RUNG wire#powerrail
      I_Contact( "PUMP" )
      Contact( "ELECTODE_DI5" )
      S_Coil( "HMI".FAIL_EL5 )
   END_RUNG
   // the same network as SCL:
   IF NOT "PUMP" AND "ELECTODE_DI5" THEN "HMI".FAIL_EL5 := TRUE; END_IF;
END_REGION

REGION Network 7: ELEKTRODE 6 ALARM
   RUNG wire#powerrail
      I_Contact( "PUMP" )
      Contact( "ELECTODE_DI6" )
      S_Coil( "HMI".FAIL_EL6 )
   END_RUNG
   // the same network as SCL:
   IF NOT "PUMP" AND "ELECTODE_DI6" THEN "HMI".FAIL_EL6 := TRUE; END_IF;
END_REGION

REGION Network 8: ELEKTRODE 7 ALARM
   RUNG wire#powerrail
      I_Contact( "PUMP" )
      Contact( "ELECTODE_DI7" )
      S_Coil( "HMI".FAIL_EL7 )
   END_RUNG
   // the same network as SCL:
   IF NOT "PUMP" AND "ELECTODE_DI7" THEN "HMI".FAIL_EL7 := TRUE; END_IF;
END_REGION

REGION Network 9: ELEKTRODE 8 ALARM
   RUNG wire#powerrail
      I_Contact( "PUMP" )
      Contact( "ELECTODE_DI8" )
      S_Coil( "HMI".FAIL_EL8 )
   END_RUNG
   // the same network as SCL:
   IF NOT "PUMP" AND "ELECTODE_DI8" THEN "HMI".FAIL_EL8 := TRUE; END_IF;
END_REGION

REGION Network 10
   RUNG wire#powerrail
      I_Contact( "PUMP" )
      S_Coil( "HMI".PUMP_STOP )
   END_RUNG
   // the same network as SCL:
   IF NOT "PUMP" THEN "HMI".PUMP_STOP := TRUE; END_IF;
END_REGION

REGION Network 11
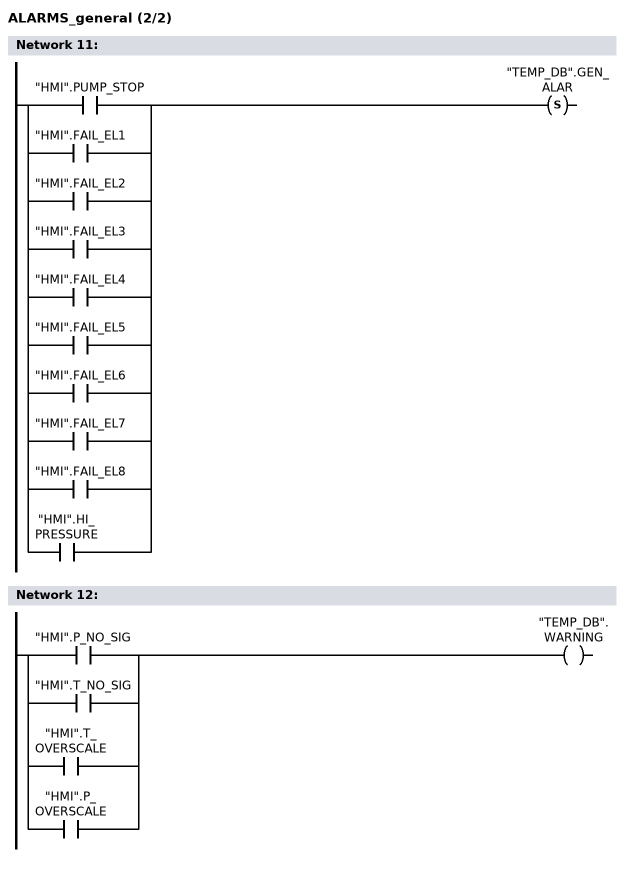
   RUNG wire#powerrail
      Contact( "HMI".PUMP_STOP )
      wire#w1
      S_Coil( "TEMP_DB".GEN_ALAR )
   END_RUNG
   RUNG wire#powerrail
      Contact( "HMI".FAIL_EL1 )
   END_RUNG wire#w1
   RUNG wire#powerrail
      Contact( "HMI".FAIL_EL2 )
   END_RUNG wire#w1
   RUNG wire#powerrail
      Contact( "HMI".FAIL_EL3 )
   END_RUNG wire#w1
   RUNG wire#powerrail
      Contact( "HMI".FAIL_EL4 )
   END_RUNG wire#w1
   RUNG wire#powerrail
      Contact( "HMI".FAIL_EL5 )
   END_RUNG wire#w1
   RUNG wire#powerrail
      Contact( "HMI".FAIL_EL6 )
   END_RUNG wire#w1
   RUNG wire#powerrail
      Contact( "HMI".FAIL_EL7 )
   END_RUNG wire#w1
   RUNG wire#powerrail
      Contact( "HMI".FAIL_EL8 )
   END_RUNG wire#w1
   RUNG wire#powerrail
      Contact( "HMI".HI_PRESSURE )
   END_RUNG wire#w1
   // the same network as SCL:
   IF "HMI".PUMP_STOP OR "HMI".FAIL_EL1 OR "HMI".FAIL_EL2 OR "HMI".FAIL_EL3 OR "HMI".FAIL_EL4 OR "HMI".FAIL_EL5 OR "HMI".FAIL_EL6 OR "HMI".FAIL_EL7 OR "HMI".FAIL_EL8 OR "HMI".HI_PRESSURE THEN
       "TEMP_DB".GEN_ALAR := TRUE;
   END_IF;
END_REGION

REGION Network 12
   RUNG wire#powerrail
      Contact( "HMI".P_NO_SIG )
      wire#w1
      Coil( "TEMP_DB".WARNING )
   END_RUNG
   RUNG wire#powerrail
      Contact( "HMI".T_NO_SIG )
   END_RUNG wire#w1
   RUNG wire#powerrail
      Contact( "HMI".T_OVERSCALE )
   END_RUNG wire#w1
   RUNG wire#powerrail
      Contact( "HMI".P_OVERSCALE )
   END_RUNG wire#w1
   // the same network as SCL:
   "TEMP_DB".WARNING := "HMI".P_NO_SIG OR "HMI".T_NO_SIG OR "HMI".T_OVERSCALE OR "HMI".P_OVERSCALE;
END_REGION
END_FUNCTION

FUNCTION "ALARMS_MAIN" : Void   // FC10, LAD
{ S7_Optimized_Access := 'TRUE' }
VERSION : 0.1
   VAR_TEMP   // added for the SCL form of the ladder/FBD networks
      _w1 : Bool;
   END_VAR
BEGIN

REGION Network 1
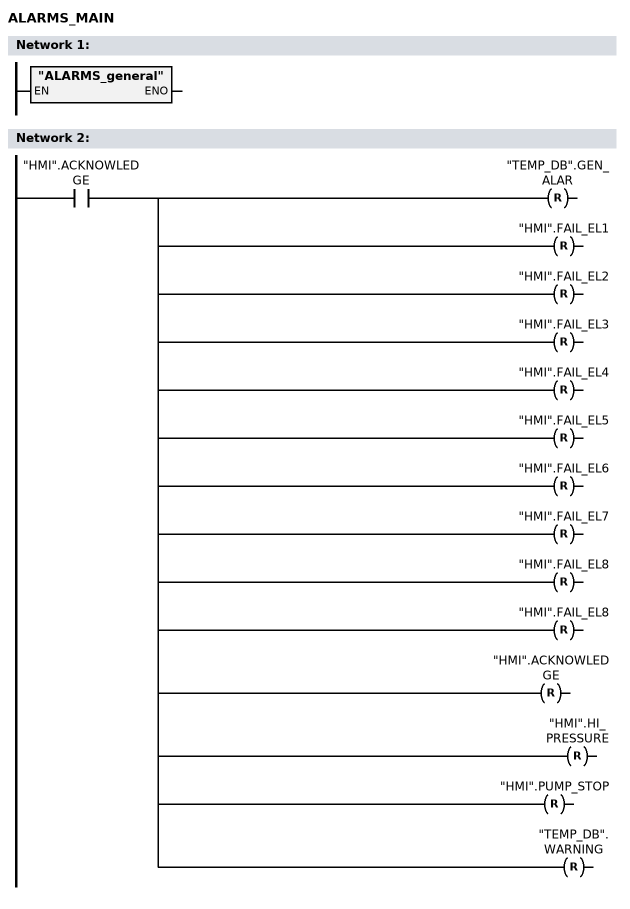
   RUNG wire#powerrail
      "ALARMS_general"()
   END_RUNG
   // the same network as SCL:
   "ALARMS_general"();
END_REGION

REGION Network 2
   RUNG wire#powerrail
      Contact( "HMI".ACKNOWLEDGE )
      wire#w1
      R_Coil( "TEMP_DB".GEN_ALAR )
   END_RUNG
   RUNG wire#w1
      R_Coil( "HMI".FAIL_EL1 )
   END_RUNG
   RUNG wire#w1
      R_Coil( "HMI".FAIL_EL2 )
   END_RUNG
   RUNG wire#w1
      R_Coil( "HMI".FAIL_EL3 )
   END_RUNG
   RUNG wire#w1
      R_Coil( "HMI".FAIL_EL4 )
   END_RUNG
   RUNG wire#w1
      R_Coil( "HMI".FAIL_EL5 )
   END_RUNG
   RUNG wire#w1
      R_Coil( "HMI".FAIL_EL6 )
   END_RUNG
   RUNG wire#w1
      R_Coil( "HMI".FAIL_EL7 )
   END_RUNG
   RUNG wire#w1
      R_Coil( "HMI".FAIL_EL8 )
   END_RUNG
   RUNG wire#w1
      R_Coil( "HMI".FAIL_EL8 )
   END_RUNG
   RUNG wire#w1
      R_Coil( "HMI".ACKNOWLEDGE )
   END_RUNG
   RUNG wire#w1
      R_Coil( "HMI".HI_PRESSURE )
   END_RUNG
   RUNG wire#w1
      R_Coil( "HMI".PUMP_STOP )
   END_RUNG
   RUNG wire#w1
      R_Coil( "TEMP_DB".WARNING )
   END_RUNG
   // the same network as SCL:
   IF "HMI".ACKNOWLEDGE THEN
       "TEMP_DB".GEN_ALAR := FALSE;
       "HMI".FAIL_EL1 := FALSE;
       "HMI".FAIL_EL2 := FALSE;
       "HMI".FAIL_EL3 := FALSE;
       "HMI".FAIL_EL4 := FALSE;
       "HMI".FAIL_EL5 := FALSE;
       "HMI".FAIL_EL6 := FALSE;
       "HMI".FAIL_EL7 := FALSE;
       "HMI".FAIL_EL8 := FALSE;
       "HMI".FAIL_EL8 := FALSE;
   END_IF;
   #_w1 := "HMI".ACKNOWLEDGE;
   IF #_w1 THEN
       "HMI".ACKNOWLEDGE := FALSE;
       "HMI".HI_PRESSURE := FALSE;
       "HMI".PUMP_STOP := FALSE;
       "TEMP_DB".WARNING := FALSE;
   END_IF;
END_REGION
END_FUNCTION

FUNCTION "TRANSLATE" : Void   // FC11, SCL
{ S7_Optimized_Access := 'TRUE' }
VERSION : 0.1
BEGIN
   (******************** REG 0 **************************)
   "BUFFER".DATA[0].%X0 := "HMI".PUMP_STOP;    (* WHEN PUMP SWITCHED OFF IT WILL BE TRUE*)
   "BUFFER".DATA[0].%X1 := "HMI".HI_PRESSURE;  (* TRUE WHEN PRESSEURE VERY HIGH *)
   "BUFFER".DATA[0].%X2 := "HMI".FAIL_EL1;     (* WHEN PROBLEM WITH ELEKTRODE 1     *)
   "BUFFER".DATA[0].%X3 := "HMI".FAIL_EL2;     (* WHEN PROBLEM WITH ELEKTRODE 2     *)
   "BUFFER".DATA[0].%X4 := "HMI".FAIL_EL3;     (* WHEN PROBLEM WITH ELEKTRODE 3     *)
   "BUFFER".DATA[0].%X5 := "HMI".FAIL_EL4;
   "BUFFER".DATA[0].%X6 := "HMI".FAIL_EL5;
   "BUFFER".DATA[0].%X7 := "HMI".FAIL_EL6;
   "BUFFER".DATA[0].%X8 := "HMI".FAIL_EL7;
   "BUFFER".DATA[0].%X9 := "HMI".FAIL_EL8;
   "HMI".ACKNOWLEDGE := "BUFFER".DATA[0].%X10;
   "HMI".ELEC_OFF1 := "BUFFER".DATA[0].%X11;   (* IGNORING ELECTRODE1 *)
   "HMI".ELEC_OFF2 := "BUFFER".DATA[0].%X12;   (* IGNORING ELECTRODE2 *)
   "HMI".ELEC_OFF3 := "BUFFER".DATA[0].%X13;   (* IGNORING ELECTRODE3 *)
   "HMI".ELEC_OFF4 := "BUFFER".DATA[0].%X14;   (* IGNORING ELECTRODE4 *)
   "HMI".ELEC_OFF5 := "BUFFER".DATA[0].%X15;   (* IGNORING ELECTRODE5 *)
   (************* REG 1  ******************)
   "HMI".ELEC_OFF6 := "BUFFER".DATA[1].%X0;    (* IGNORING ELECTRODE6 *)
   "HMI".ELEC_OFF7 := "BUFFER".DATA[1].%X1;    (* IGNORING ELECTRODE7 *)
   "HMI".ELEC_OFF8 := "BUFFER".DATA[1].%X2;    (* IGNORING ELECTRODE8 *)
   "HMI".DO_TEST := "BUFFER".DATA[1].%X3;      (*FOR TESTING DISCRET OUTPUTS*)
   "HMI".T_SIMUL := "BUFFER".DATA[1].%X4;
   "HMI".P_SIMUL := "BUFFER".DATA[1].%X5;
   "BUFFER".DATA[1].%X6 := "HMI".T_NO_SIG;
   "BUFFER".DATA[1].%X7 := "HMI".P_NO_SIG;
   "BUFFER".DATA[1].%X8 := "HMI".T_OVERSCALE;
   "BUFFER".DATA[1].%X9 := "HMI".P_OVERSCALE;




   (****************************** REG 2 - 3 *********************************************)
   "BUFFER".DATA[2].%X0 := "PUMP";
   "BUFFER".DATA[2].%X1 := "AUTO_MAN";
   "BUFFER".DATA[2].%X2 := "ELECTODE_DI1";
   "BUFFER".DATA[2].%X3 := "ELECTODE_DI2";
   "BUFFER".DATA[2].%X4 := "ELECTODE_DI3";
   "BUFFER".DATA[2].%X5 := "ELECTODE_DI4";
   "BUFFER".DATA[2].%X6 := "ELECTODE_DI5";
   "BUFFER".DATA[2].%X7 := "ELECTODE_DI6";
   "BUFFER".DATA[2].%X8 := "ELECTODE_DI7";
   "BUFFER".DATA[2].%X9 := "ELECTODE_DI8";

   IF "HMI".DO_TEST THEN
       "ELECTR_DO_1" := "BUFFER".DATA[2].%X10;
       "ELECTR_DO_2" := "BUFFER".DATA[2].%X11;
       "ELECTR_DO_3" := "BUFFER".DATA[2].%X12;
       "ELECTR_DO_4" := "BUFFER".DATA[2].%X13;
       "ELECTR_DO_5" := "BUFFER".DATA[2].%X14;
       "ELECTR_DO_6" := "BUFFER".DATA[2].%X15;
       "ELECTR_DO_7" := "BUFFER".DATA[3].%X0;
       "ELECTR_DO_8" := "BUFFER".DATA[3].%X1;
   END_IF;
   (********************************* REG 3 ***************************************************)
END_FUNCTION

ORGANIZATION_BLOCK "Main"   // OB1, LAD, ProgramCycle
TITLE = "Main Program Sweep (Cycle)"
{ S7_Optimized_Access := 'TRUE' }
VERSION : 0.1
   VAR_INPUT
      Initial_Call : Bool;   // Initial call of this OB
      Remanence : Bool;   // =True, if remanent data are available
   END_VAR
   VAR_TEMP   // added for the SCL form of the ladder/FBD networks
      _w1 : Bool;
   END_VAR
BEGIN

REGION Network 1
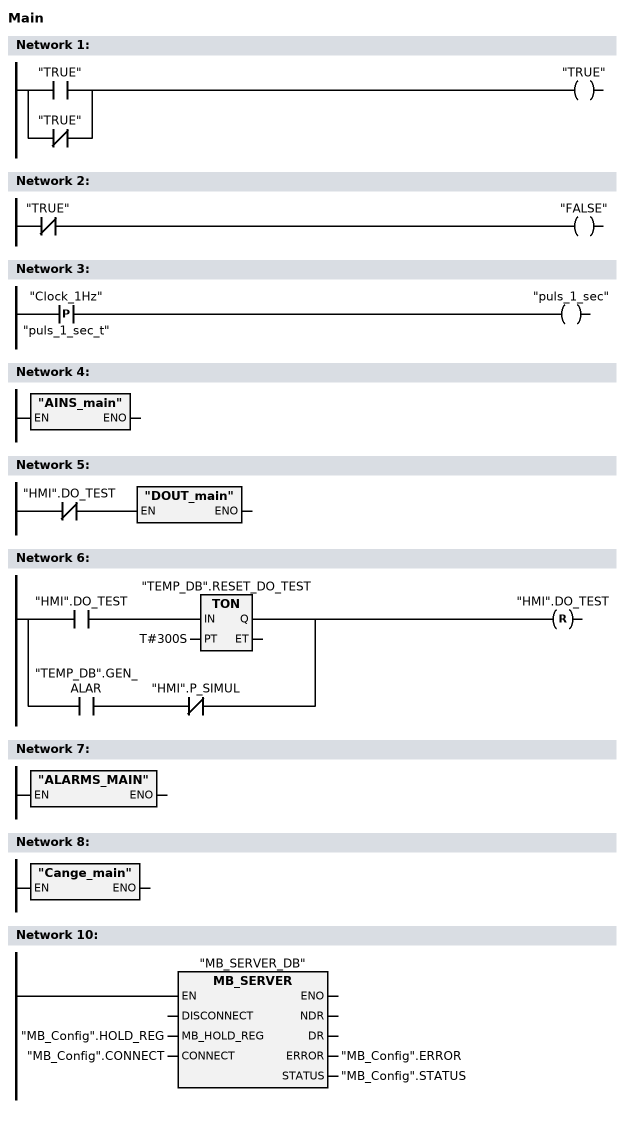
   RUNG wire#powerrail
      Contact( "TRUE" )
      wire#w1
      Coil( "TRUE" )
   END_RUNG
   RUNG wire#powerrail
      I_Contact( "TRUE" )
   END_RUNG wire#w1
   // the same network as SCL:
   "TRUE" := "TRUE" OR NOT "TRUE";
END_REGION

REGION Network 2
   RUNG wire#powerrail
      I_Contact( "TRUE" )
      Coil( "FALSE" )
   END_RUNG
   // the same network as SCL:
   "FALSE" := NOT "TRUE";
END_REGION

REGION Network 3
   RUNG wire#powerrail
      P_Contact(operand := "Clock_1Hz", bit := "puls_1_sec_t")
      Coil( "puls_1_sec" )
   END_RUNG
   // the same network as SCL:
   #_w1 := "Clock_1Hz" AND NOT "puls_1_sec_t";   // rising edge of "Clock_1Hz"
   "puls_1_sec_t" := "Clock_1Hz";
   "puls_1_sec" := #_w1;
END_REGION

REGION Network 4
   RUNG wire#powerrail
      "AINS_main"()
   END_RUNG
   // the same network as SCL:
   "AINS_main"();
END_REGION

REGION Network 5
   RUNG wire#powerrail
      I_Contact( "HMI".DO_TEST )
      "DOUT_main"()
   END_RUNG
   // the same network as SCL:
   IF NOT "HMI".DO_TEST THEN "DOUT_main"(); END_IF;
END_REGION

REGION Network 6
   "TEMP_DB".RESET_DO_TEST.TON(IN := "HMI".DO_TEST, PT := T#300S);
   IF "TEMP_DB".RESET_DO_TEST.Q OR ("TEMP_DB".GEN_ALAR AND NOT "HMI".P_SIMUL) THEN
       "HMI".DO_TEST := FALSE;
   END_IF;
END_REGION

REGION Network 7
   RUNG wire#powerrail
      "ALARMS_MAIN"()
   END_RUNG
   // the same network as SCL:
   "ALARMS_MAIN"();
END_REGION

REGION Network 8
   RUNG wire#powerrail
      "Cange_main"()
   END_RUNG
   // the same network as SCL:
   "Cange_main"();
END_REGION

REGION Network 10
   "MB_SERVER_DB"(MB_HOLD_REG := "MB_Config".HOLD_REG,   // MB_SERVER
                  CONNECT := "MB_Config".CONNECT,
                  ERROR => "MB_Config".ERROR,
                  STATUS => "MB_Config".STATUS);
END_REGION
END_ORGANIZATION_BLOCK